PROGRAM P1_03_Alarms
VAR
	iActive				:INT;
	iAck				:INT;
	iRaise				:INT;
	
	bAlarmActive		:BOOL;
	bWarningActive		:BOOL;
	
	bAckAll				:BOOL;

	TON_Ack				:TON;
	TON_AlarmOK			:TON;

	TON_Alarm			:ARRAY[0..39] OF TON;
	
	
	
	
	Simulation	:BOOL;
	bTest: BOOL;
END_VAR
VAR // added by the converter: edge detectors and wires of the graphical bodies
    _rt1, _rt2, _rt3 : R_TRIG;
END_VAR

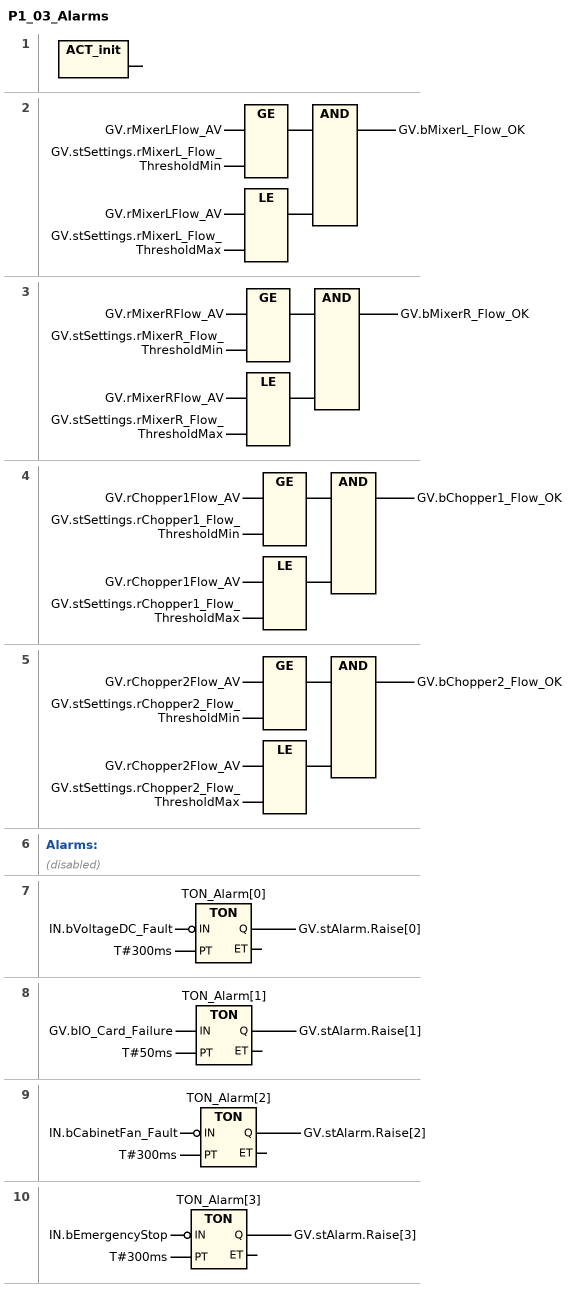
// NETWORK 1
ACT_init();

// NETWORK 2
GV.bMixerL_Flow_OK := GV.rMixerLFlow_AV >= GV.stSettings.rMixerL_Flow_ThresholdMin AND GV.rMixerLFlow_AV <= GV.stSettings.rMixerL_Flow_ThresholdMax;

// NETWORK 3
GV.bMixerR_Flow_OK := GV.rMixerRFlow_AV >= GV.stSettings.rMixerR_Flow_ThresholdMin AND GV.rMixerRFlow_AV <= GV.stSettings.rMixerR_Flow_ThresholdMax;

// NETWORK 4
GV.bChopper1_Flow_OK := GV.rChopper1Flow_AV >= GV.stSettings.rChopper1_Flow_ThresholdMin AND GV.rChopper1Flow_AV <= GV.stSettings.rChopper1_Flow_ThresholdMax;

// NETWORK 5
GV.bChopper2_Flow_OK := GV.rChopper2Flow_AV >= GV.stSettings.rChopper2_Flow_ThresholdMin AND GV.rChopper2Flow_AV <= GV.stSettings.rChopper2_Flow_ThresholdMax;

// NETWORK 6 (disabled)
// label: Alarms

// NETWORK 7
TON_Alarm[0](IN := NOT IN.bVoltageDC_Fault, PT := T#300ms); // TON
GV.stAlarm.Raise[0] := TON_Alarm[0].Q;

// NETWORK 8
TON_Alarm[1](IN := GV.bIO_Card_Failure, PT := T#50ms); // TON
GV.stAlarm.Raise[1] := TON_Alarm[1].Q;

// NETWORK 9
TON_Alarm[2](IN := NOT IN.bCabinetFan_Fault, PT := T#300ms); // TON
GV.stAlarm.Raise[2] := TON_Alarm[2].Q;

// NETWORK 10
TON_Alarm[3](IN := NOT IN.bEmergencyStop, PT := T#300ms); // TON
GV.stAlarm.Raise[3] := TON_Alarm[3].Q;

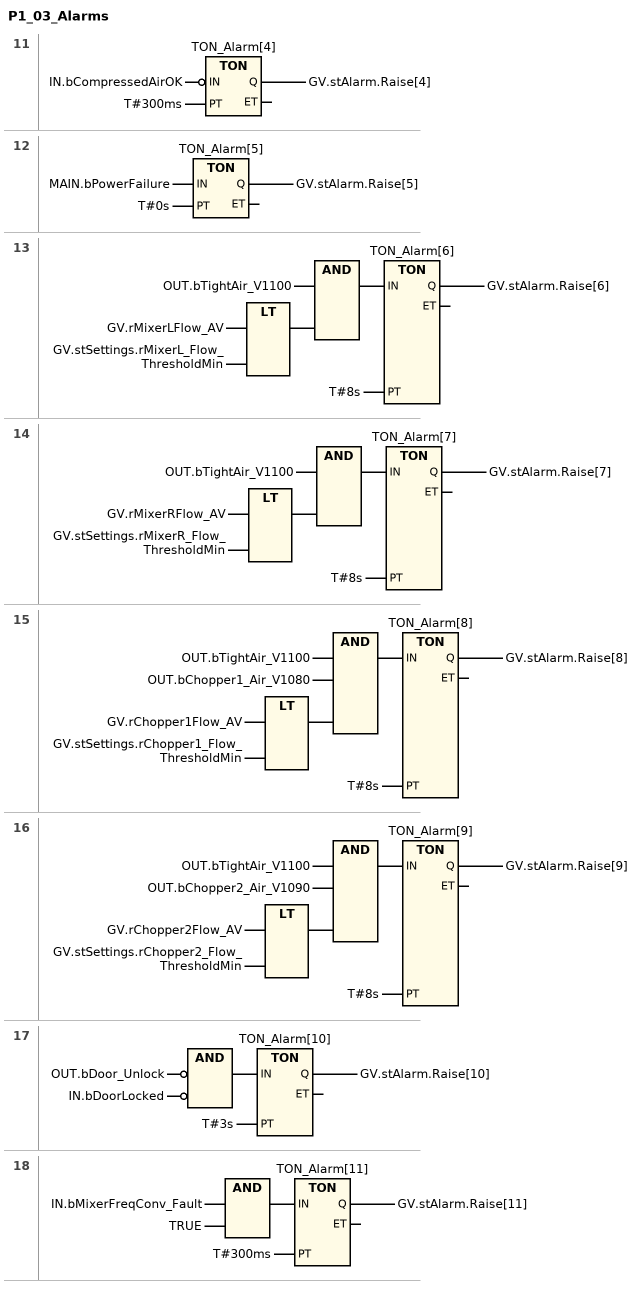
// NETWORK 11
TON_Alarm[4](IN := NOT IN.bCompressedAirOK, PT := T#300ms); // TON
GV.stAlarm.Raise[4] := TON_Alarm[4].Q;

// NETWORK 12
TON_Alarm[5](IN := MAIN.bPowerFailure, PT := T#0s); // TON
GV.stAlarm.Raise[5] := TON_Alarm[5].Q;

// NETWORK 13
TON_Alarm[6](IN := OUT.bTightAir_V1100 AND GV.rMixerLFlow_AV < GV.stSettings.rMixerL_Flow_ThresholdMin, PT := T#8s); // TON
GV.stAlarm.Raise[6] := TON_Alarm[6].Q;

// NETWORK 14
TON_Alarm[7](IN := OUT.bTightAir_V1100 AND GV.rMixerRFlow_AV < GV.stSettings.rMixerR_Flow_ThresholdMin, PT := T#8s); // TON
GV.stAlarm.Raise[7] := TON_Alarm[7].Q;

// NETWORK 15
TON_Alarm[8](IN := OUT.bTightAir_V1100 AND OUT.bChopper1_Air_V1080 AND GV.rChopper1Flow_AV < GV.stSettings.rChopper1_Flow_ThresholdMin, PT := T#8s); // TON
GV.stAlarm.Raise[8] := TON_Alarm[8].Q;

// NETWORK 16
TON_Alarm[9](IN := OUT.bTightAir_V1100 AND OUT.bChopper2_Air_V1090 AND GV.rChopper2Flow_AV < GV.stSettings.rChopper2_Flow_ThresholdMin, PT := T#8s); // TON
GV.stAlarm.Raise[9] := TON_Alarm[9].Q;

// NETWORK 17
TON_Alarm[10](IN := NOT OUT.bDoor_Unlock AND NOT IN.bDoorLocked, PT := T#3s); // TON
GV.stAlarm.Raise[10] := TON_Alarm[10].Q;

// NETWORK 18
TON_Alarm[11](IN := IN.bMixerFreqConv_Fault AND TRUE, PT := T#300ms); // TON
GV.stAlarm.Raise[11] := TON_Alarm[11].Q;

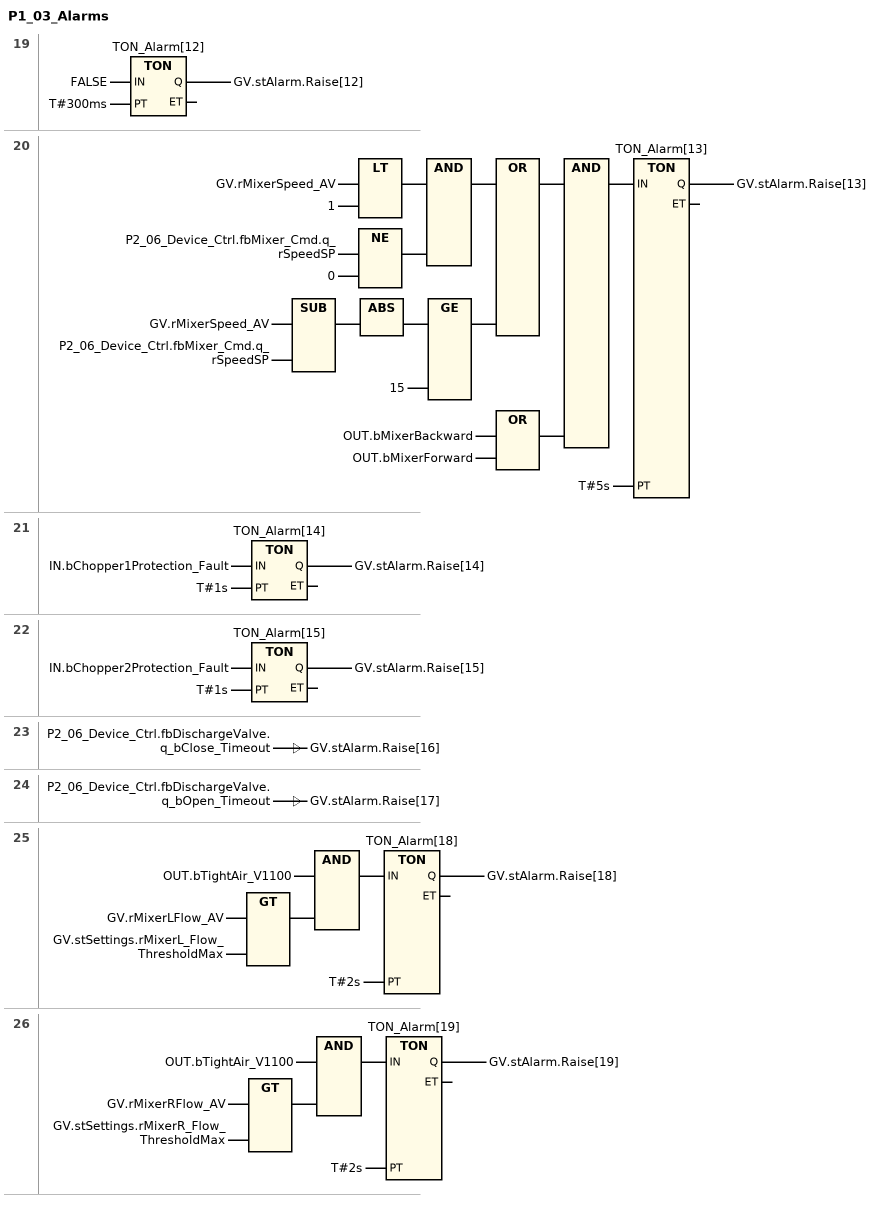
// NETWORK 19
TON_Alarm[12](IN := FALSE, PT := T#300ms); // TON
GV.stAlarm.Raise[12] := TON_Alarm[12].Q;

// NETWORK 20
TON_Alarm[13](IN := (GV.rMixerSpeed_AV < 1 AND P2_06_Device_Ctrl.fbMixer_Cmd.q_rSpeedSP <> 0 OR ABS(GV.rMixerSpeed_AV - P2_06_Device_Ctrl.fbMixer_Cmd.q_rSpeedSP) >= 15) AND (OUT.bMixerBackward OR OUT.bMixerForward), PT := T#5s); // TON
GV.stAlarm.Raise[13] := TON_Alarm[13].Q;

// NETWORK 21
TON_Alarm[14](IN := IN.bChopper1Protection_Fault, PT := T#1s); // TON
GV.stAlarm.Raise[14] := TON_Alarm[14].Q;

// NETWORK 22
TON_Alarm[15](IN := IN.bChopper2Protection_Fault, PT := T#1s); // TON
GV.stAlarm.Raise[15] := TON_Alarm[15].Q;

// NETWORK 23
_rt1(CLK := P2_06_Device_Ctrl.fbDischargeValve.q_bClose_Timeout);
GV.stAlarm.Raise[16] := _rt1.Q;

// NETWORK 24
_rt2(CLK := P2_06_Device_Ctrl.fbDischargeValve.q_bOpen_Timeout);
GV.stAlarm.Raise[17] := _rt2.Q;

// NETWORK 25
TON_Alarm[18](IN := OUT.bTightAir_V1100 AND GV.rMixerLFlow_AV > GV.stSettings.rMixerL_Flow_ThresholdMax, PT := T#2s); // TON
GV.stAlarm.Raise[18] := TON_Alarm[18].Q;

// NETWORK 26
TON_Alarm[19](IN := OUT.bTightAir_V1100 AND GV.rMixerRFlow_AV > GV.stSettings.rMixerR_Flow_ThresholdMax, PT := T#2s); // TON
GV.stAlarm.Raise[19] := TON_Alarm[19].Q;

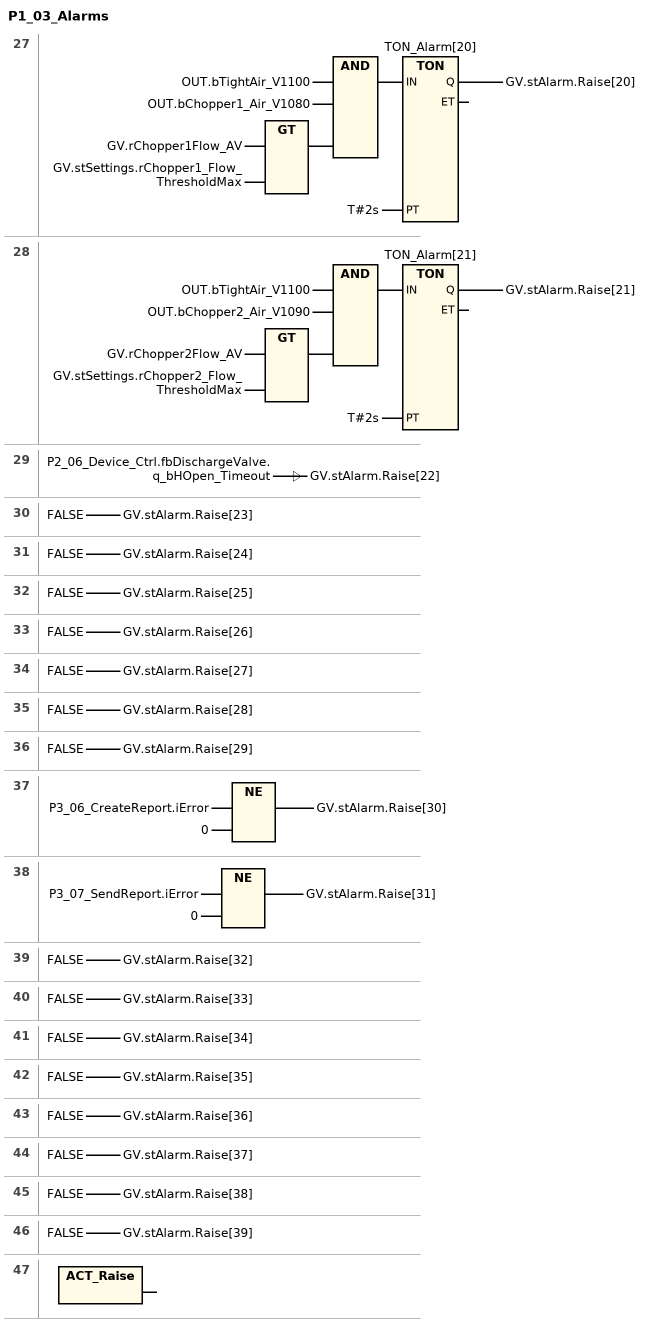
// NETWORK 27
TON_Alarm[20](IN := OUT.bTightAir_V1100 AND OUT.bChopper1_Air_V1080 AND GV.rChopper1Flow_AV > GV.stSettings.rChopper1_Flow_ThresholdMax, PT := T#2s); // TON
GV.stAlarm.Raise[20] := TON_Alarm[20].Q;

// NETWORK 28
TON_Alarm[21](IN := OUT.bTightAir_V1100 AND OUT.bChopper2_Air_V1090 AND GV.rChopper2Flow_AV > GV.stSettings.rChopper2_Flow_ThresholdMax, PT := T#2s); // TON
GV.stAlarm.Raise[21] := TON_Alarm[21].Q;

// NETWORK 29
_rt3(CLK := P2_06_Device_Ctrl.fbDischargeValve.q_bHOpen_Timeout);
GV.stAlarm.Raise[22] := _rt3.Q;

// NETWORK 30
GV.stAlarm.Raise[23] := FALSE;

// NETWORK 31
GV.stAlarm.Raise[24] := FALSE;

// NETWORK 32
GV.stAlarm.Raise[25] := FALSE;

// NETWORK 33
GV.stAlarm.Raise[26] := FALSE;

// NETWORK 34
GV.stAlarm.Raise[27] := FALSE;

// NETWORK 35
GV.stAlarm.Raise[28] := FALSE;

// NETWORK 36
GV.stAlarm.Raise[29] := FALSE;

// NETWORK 37
GV.stAlarm.Raise[30] := P3_06_CreateReport.iError <> 0;

// NETWORK 38
GV.stAlarm.Raise[31] := P3_07_SendReport.iError <> 0;

// NETWORK 39
GV.stAlarm.Raise[32] := FALSE;

// NETWORK 40
GV.stAlarm.Raise[33] := FALSE;

// NETWORK 41
GV.stAlarm.Raise[34] := FALSE;

// NETWORK 42
GV.stAlarm.Raise[35] := FALSE;

// NETWORK 43
GV.stAlarm.Raise[36] := FALSE;

// NETWORK 44
GV.stAlarm.Raise[37] := FALSE;

// NETWORK 45
GV.stAlarm.Raise[38] := FALSE;

// NETWORK 46
GV.stAlarm.Raise[39] := FALSE;

// NETWORK 47
ACT_Raise();

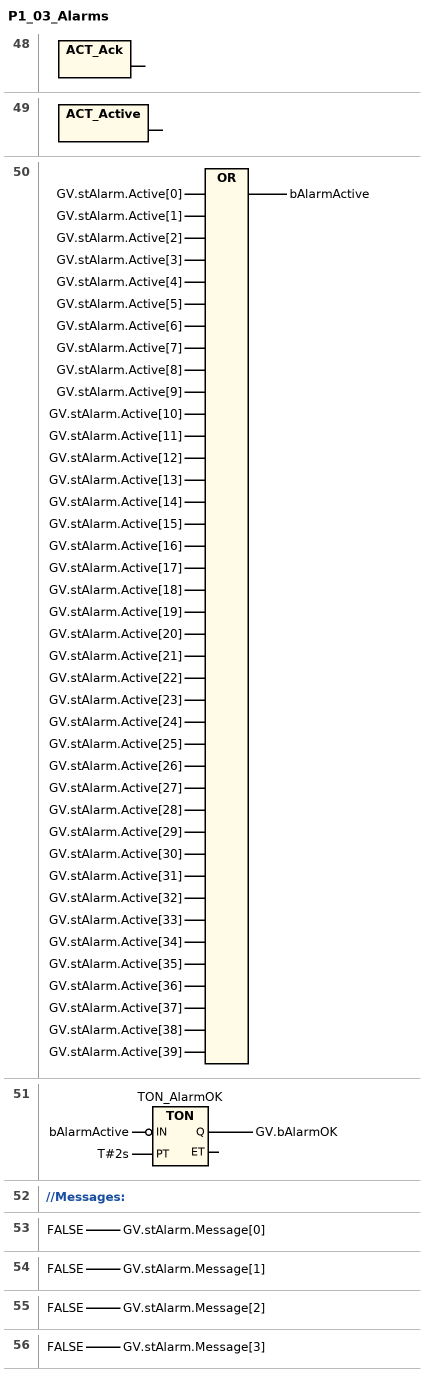
// NETWORK 48
ACT_Ack();

// NETWORK 49
ACT_Active();

// NETWORK 50
bAlarmActive := GV.stAlarm.Active[0] OR GV.stAlarm.Active[1] OR GV.stAlarm.Active[2] OR GV.stAlarm.Active[3] OR GV.stAlarm.Active[4] OR GV.stAlarm.Active[5] OR GV.stAlarm.Active[6] OR GV.stAlarm.Active[7] OR GV.stAlarm.Active[8] OR GV.stAlarm.Active[9] OR GV.stAlarm.Active[10] OR GV.stAlarm.Active[11] OR GV.stAlarm.Active[12] OR GV.stAlarm.Active[13] OR GV.stAlarm.Active[14] OR GV.stAlarm.Active[15] OR GV.stAlarm.Active[16] OR GV.stAlarm.Active[17] OR GV.stAlarm.Active[18] OR GV.stAlarm.Active[19] OR GV.stAlarm.Active[20] OR GV.stAlarm.Active[21] OR GV.stAlarm.Active[22] OR GV.stAlarm.Active[23] OR GV.stAlarm.Active[24] OR GV.stAlarm.Active[25] OR GV.stAlarm.Active[26] OR GV.stAlarm.Active[27] OR GV.stAlarm.Active[28] OR GV.stAlarm.Active[29] OR GV.stAlarm.Active[30] OR GV.stAlarm.Active[31] OR GV.stAlarm.Active[32] OR GV.stAlarm.Active[33] OR GV.stAlarm.Active[34] OR GV.stAlarm.Active[35] OR GV.stAlarm.Active[36] OR GV.stAlarm.Active[37] OR GV.stAlarm.Active[38] OR GV.stAlarm.Active[39];

// NETWORK 51
TON_AlarmOK(IN := NOT bAlarmActive, PT := T#2s); // TON
GV.bAlarmOK := TON_AlarmOK.Q;

// NETWORK 52
// label: //Messages

// NETWORK 53
GV.stAlarm.Message[0] := FALSE;

// NETWORK 54
GV.stAlarm.Message[1] := FALSE;

// NETWORK 55
GV.stAlarm.Message[2] := FALSE;

// NETWORK 56
GV.stAlarm.Message[3] := FALSE;

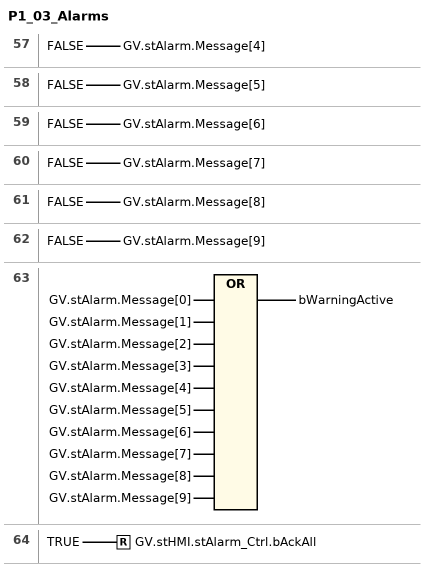
// NETWORK 57
GV.stAlarm.Message[4] := FALSE;

// NETWORK 58
GV.stAlarm.Message[5] := FALSE;

// NETWORK 59
GV.stAlarm.Message[6] := FALSE;

// NETWORK 60
GV.stAlarm.Message[7] := FALSE;

// NETWORK 61
GV.stAlarm.Message[8] := FALSE;

// NETWORK 62
GV.stAlarm.Message[9] := FALSE;

// NETWORK 63
bWarningActive := GV.stAlarm.Message[0] OR GV.stAlarm.Message[1] OR GV.stAlarm.Message[2] OR GV.stAlarm.Message[3] OR GV.stAlarm.Message[4] OR GV.stAlarm.Message[5] OR GV.stAlarm.Message[6] OR GV.stAlarm.Message[7] OR GV.stAlarm.Message[8] OR GV.stAlarm.Message[9];

// NETWORK 64
GV.stHMI.stAlarm_Ctrl.bAckAll R= TRUE;

ACTION ACT_Ack:
FOR iAck:=0 TO 99 DO
	IF GV.stAlarm.Alarm[iAck].eConfirmationState = 3 OR GV.stHMI.stAlarm_Ctrl.bAckAll THEN
		GV.stAlarm.Alarm[iAck].Clear(0,1);
	END_IF
	
	IF GV.stAlarm.Warning[iAck].bRaised AND NOT GV.stAlarm.Message[iAck] THEN
		GV.stAlarm.Warning[iAck].Clear(0,1);
	END_IF
END_FOR
END_ACTION

ACTION ACT_Active:
FOR iActive:=0 TO 99 DO
	GV.stAlarm.Active[iActive]:=GV.stAlarm.Alarm[iActive].bActive;
END_FOR
END_ACTION

ACTION ACT_Init:
IF MAIN.bFirstCycle THEN
	//Critical
	GV.stAlarm.Alarm[0].CreateEx(TC_EVENTS.Alarms.AlarmsEvent1,1,0);
	GV.stAlarm.Alarm[1].CreateEx(TC_EVENTS.Alarms.AlarmsEvent2,1,0);
	GV.stAlarm.Alarm[2].CreateEx(TC_EVENTS.Alarms.AlarmsEvent3,1,0);
	GV.stAlarm.Alarm[3].CreateEx(TC_EVENTS.Alarms.AlarmsEvent4,1,0);
	GV.stAlarm.Alarm[4].CreateEx(TC_EVENTS.Alarms.AlarmsEvent5,1,0);
	GV.stAlarm.Alarm[5].CreateEx(TC_EVENTS.Alarms.AlarmsEvent6,1,0);
	GV.stAlarm.Alarm[6].CreateEx(TC_EVENTS.Alarms.AlarmsEvent7,1,0);
	GV.stAlarm.Alarm[7].CreateEx(TC_EVENTS.Alarms.AlarmsEvent8,1,0);
	GV.stAlarm.Alarm[8].CreateEx(TC_EVENTS.Alarms.AlarmsEvent9,1,0);
	GV.stAlarm.Alarm[9].CreateEx(TC_EVENTS.Alarms.AlarmsEvent10,1,0);
	GV.stAlarm.Alarm[10].CreateEx(TC_EVENTS.Alarms.AlarmsEvent11,1,0);
	GV.stAlarm.Alarm[11].CreateEx(TC_EVENTS.Alarms.AlarmsEvent12,1,0);
	GV.stAlarm.Alarm[12].CreateEx(TC_EVENTS.Alarms.AlarmsEvent13,1,0);
	GV.stAlarm.Alarm[13].CreateEx(TC_EVENTS.Alarms.AlarmsEvent14,1,0);
	GV.stAlarm.Alarm[14].CreateEx(TC_EVENTS.Alarms.AlarmsEvent15,1,0);
	GV.stAlarm.Alarm[15].CreateEx(TC_EVENTS.Alarms.AlarmsEvent16,1,0);
	GV.stAlarm.Alarm[16].CreateEx(TC_EVENTS.Alarms.AlarmsEvent17,1,0);
	GV.stAlarm.Alarm[17].CreateEx(TC_EVENTS.Alarms.AlarmsEvent18,1,0);
	GV.stAlarm.Alarm[18].CreateEx(TC_EVENTS.Alarms.AlarmsEvent19,1,0);
	GV.stAlarm.Alarm[19].CreateEx(TC_EVENTS.Alarms.AlarmsEvent20,1,0);
	GV.stAlarm.Alarm[20].CreateEx(TC_EVENTS.Alarms.AlarmsEvent21,1,0);
	GV.stAlarm.Alarm[21].CreateEx(TC_EVENTS.Alarms.AlarmsEvent22,1,0);
	GV.stAlarm.Alarm[22].CreateEx(TC_EVENTS.Alarms.AlarmsEvent23,1,0);
	GV.stAlarm.Alarm[23].CreateEx(TC_EVENTS.Alarms.AlarmsEvent24,1,0);
	GV.stAlarm.Alarm[24].CreateEx(TC_EVENTS.Alarms.AlarmsEvent25,1,0);
	GV.stAlarm.Alarm[25].CreateEx(TC_EVENTS.Alarms.AlarmsEvent26,1,0);
	GV.stAlarm.Alarm[26].CreateEx(TC_EVENTS.Alarms.AlarmsEvent27,1,0);
	GV.stAlarm.Alarm[27].CreateEx(TC_EVENTS.Alarms.AlarmsEvent28,1,0);
	GV.stAlarm.Alarm[28].CreateEx(TC_EVENTS.Alarms.AlarmsEvent29,1,0);
	GV.stAlarm.Alarm[29].CreateEx(TC_EVENTS.Alarms.AlarmsEvent30,1,0);
	GV.stAlarm.Alarm[30].CreateEx(TC_EVENTS.Alarms.AlarmsEvent31,1,0);
	GV.stAlarm.Alarm[31].CreateEx(TC_EVENTS.Alarms.AlarmsEvent32,1,0);
	GV.stAlarm.Alarm[32].CreateEx(TC_EVENTS.Alarms.AlarmsEvent33,1,0);
	GV.stAlarm.Alarm[33].CreateEx(TC_EVENTS.Alarms.AlarmsEvent34,1,0);
	GV.stAlarm.Alarm[34].CreateEx(TC_EVENTS.Alarms.AlarmsEvent35,1,0);
	GV.stAlarm.Alarm[35].CreateEx(TC_EVENTS.Alarms.AlarmsEvent36,1,0);
	GV.stAlarm.Alarm[36].CreateEx(TC_EVENTS.Alarms.AlarmsEvent37,1,0);
	GV.stAlarm.Alarm[37].CreateEx(TC_EVENTS.Alarms.AlarmsEvent38,1,0);
	GV.stAlarm.Alarm[38].CreateEx(TC_EVENTS.Alarms.AlarmsEvent39,1,0);
	GV.stAlarm.Alarm[39].CreateEx(TC_EVENTS.Alarms.AlarmsEvent40,1,0);	
END_IF
END_ACTION

ACTION ACT_Raise:
FOR iRaise:=0 TO 99 DO
	IF GV.stAlarm.Raise[iRaise] THEN
		GV.stAlarm.Alarm[iRaise].Raise(0);
	END_IF
	
	IF GV.stAlarm.Message[iRaise] THEN
		GV.stAlarm.Warning[iRaise].Raise(0);
	END_IF
END_FOR
END_ACTION

END_PROGRAM

(* stored: Version 1.1.0.1
   POU P1_03_Alarms: Id {05a3b4e5-763c-4134-adea-e0ffcecea08d}, SpecialFunc None
   Action ACT_Ack: Id {38bcc089-4166-4bc8-8e7d-87cb4ae9c08b}
   Action ACT_Active: Id {03da289e-5970-482e-a297-51b7f8397c80}
   Action ACT_Init: Id {181bf5ce-27d5-4fe3-b170-4e8cad8c1884}
   Action ACT_Raise: Id {c0adc887-b8e8-40fe-922b-74f7b64f19fc} *)
